FUNCTION_BLOCK FB_Sensor
VAR_INPUT
	lock:bool:=false;
END_VAR
VAR_OUTPUT
END_VAR
VAR
	Sensor AT %I*:BOOL:=FALSE;
	notSensor AT %I*:BOOL:=false;
	Q :BOOL;
	trigger:R_TRIG;
END_VAR

IF NOT lock THEN
	trigger(CLK:=(Sensor XOR (NOT notSensor)));
	IF trigger.Q THEN Q:=TRUE; END_IF
END_IF

METHOD isActive : BOOL
VAR_INPUT
END_VAR
IF Sensor then isActive:=true; else isActive:=false; End_if
END_METHOD

METHOD quitRising : BOOL
VAR_INPUT
END_VAR
Q:=false;
END_METHOD

METHOD wasRising : BOOL
VAR_INPUT
END_VAR
wasRising:=Q;
Q:=false;
END_METHOD

END_FUNCTION_BLOCK

(* stored: Version 1.1.0.1, ProductVersion 3.1.4022.9
   POU FB_Sensor: Id {d74e825a-653c-4340-9b40-d8020f4f45f6}, SpecialFunc None
   Method isActive: Id {d0b19cee-9c78-4c15-b332-6b44a2214aa0}
   Method quitRising: Id {a9cbc78f-c24e-4670-9390-01c922e4e188}
   Method wasRising: Id {617a1664-9f50-4ccb-8b7a-18b7444808d5} *)
